// TIA Portal project "LAP_2018_Abfuellanlage" (V14)

(* hardware
DEVICE "S7-1200-Station_1"  S7-1200 Station
   slot 0: "Baugruppenträger_0"  S7-1200 Rack  Rack  V1.0
   slot 1: "PLC_1"  CPU 1214C DC/DC/DC  6ES7 214-1AG40-0XB0  V4.2
   slot 3: "AQ 1x12BIT_1"  AQ1 signal board  6ES7 232-4HA30-0XB0  V1.0
*)

// ===== PLC "PLC_1"  CPU 1214C DC/DC/DC =====

VAR_GLOBAL   // PLC tag table "Standard-Variablentabelle"
   "System_Byte" AT %MB100 : Byte;
   "FirstScan" AT %M100.0 : Bool;
   "DiagStatusUpdate" AT %M100.1 : Bool;
   "AlwaysTRUE" AT %M100.2 : Bool;
   "AlwaysFALSE" AT %M100.3 : Bool;
   "Clock_Byte" AT %MB110 : Byte;
   "Clock_10Hz" AT %M110.0 : Bool;
   "Clock_5Hz" AT %M110.1 : Bool;
   "Clock_2.5Hz" AT %M110.2 : Bool;
   "Clock_2Hz" AT %M110.3 : Bool;
   "Clock_1.25Hz" AT %M110.4 : Bool;
   "Clock_1Hz" AT %M110.5 : Bool;
   "Clock_0.625Hz" AT %M110.6 : Bool;
   "Clock_0.5Hz" AT %M110.7 : Bool;
   "Q1" AT %Q0.0 : Bool;   // Nicht verwenden! - Nur zum Testen
   "Q2" AT %Q0.1 : Bool;   // Nicht verwenden! - Nur zum Testen
   "S1" AT %I0.0 : Bool;   // Nicht verwenden! - Nur zum Testen
   "S2" AT %I0.1 : Bool;   // Nicht verwenden! - Nur zum Testen
   "S3" AT %I0.2 : Bool;   // Nicht verwenden! - Nur zum Testen
   "S4" AT %I0.3 : Bool;   // Nicht verwenden! - Nur zum Testen
   "S5" AT %I0.4 : Bool;   // Nicht verwenden! - Nur zum Testen
   "AlleAusgänge" AT %QW0 : Word;   // Nicht löschen!
   "Q3" AT %Q0.2 : Bool;   // Nicht verwenden! - Nur zum Testen
   "Q4" AT %Q0.3 : Bool;   // Nicht verwenden! - Nur zum Testen
   "Q5" AT %Q0.4 : Bool;   // Nicht verwenden! - Nur zum Testen
   "Q6" AT %Q0.5 : Bool;   // Nicht verwenden! - Nur zum Testen
END_VAR

DATA_BLOCK "VersionInput"   // DB1
{ S7_Optimized_Access := 'FALSE' }
VERSION : 0.1
   VAR
      AutoTest : Bool;
      "Version" : String := 'LAP 2018/2 Abfuellanlage V2.0';
   END_VAR
BEGIN
END_DATA_BLOCK

DATA_BLOCK "DigInput"   // DB2
{ S7_Optimized_Access := 'FALSE' }
VERSION : 0.1
   VAR
      B1 : Bool;   // Position Flasche
      F5 : Bool;   // Motorschutzschalter
      S1 : Bool;   // Start
      S2 : Bool;   // Stop
      S3 : Bool;   // Vereinzelung
      S4 : Bool;   // Quittieren
   END_VAR
BEGIN
END_DATA_BLOCK

DATA_BLOCK "DigOutput"   // DB3
{ S7_Optimized_Access := 'FALSE' }
VERSION : 0.1
   VAR
      M1 : Bool;   // Antrieb Förderband
      K1 : Bool;   // Füllung
      K2 : Bool;   // Vereinzelung
      P1 : Bool;   // Anlage Ein
      P2 : Bool;   // Störung
   END_VAR
BEGIN
END_DATA_BLOCK

DATA_BLOCK "AnInput"   // DB4
{ S7_Optimized_Access := 'FALSE' }
VERSION : 0.1
   VAR
      PegelByte : Byte;
      PegelInt : Int;
   END_VAR
BEGIN
END_DATA_BLOCK

FUNCTION "DeleteMe" : Void   // FC1, SCL
{ S7_Optimized_Access := 'TRUE' }
VERSION : 0.1
BEGIN
   "DigOutput".K1 := "S1";
   "DigOutput".K2 := "S2";
   "DigOutput".M1 := "S3";
   "DigOutput".P1 := "S4";
   "DigOutput".P2 := "S5";

   "Q1" := "DigInput".B1;
   "Q2" := "DigInput".F5;
   "Q3" := "DigInput".S1;
   "Q4" := "DigInput".S2;
   "Q5" := "DigInput".S3;
   "Q6" := "DigInput".S4;
END_FUNCTION

FUNCTION "DatenRangieren" : Void   // FC2, SCL
{ S7_Optimized_Access := 'TRUE' }
VERSION : 0.1
BEGIN
END_FUNCTION

ORGANIZATION_BLOCK "Main"   // OB1, LAD, ProgramCycle
TITLE = "Main Program Sweep (Cycle)"
{ S7_Optimized_Access := 'TRUE' }
VERSION : 0.1
   VAR_INPUT
      Initial_Call : Bool;   // Initial call of this OB
      Remanence : Bool;   // =True, if remanent data are available
   END_VAR
BEGIN

REGION Network 1
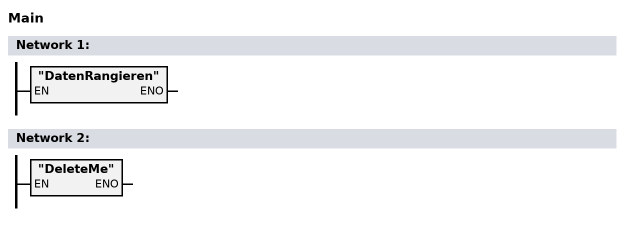
   RUNG wire#powerrail
      "DatenRangieren"()
   END_RUNG
   // the same network as SCL:
   "DatenRangieren"();
END_REGION

REGION Network 2
   RUNG wire#powerrail
      "DeleteMe"()
   END_RUNG
   // the same network as SCL:
   "DeleteMe"();
END_REGION
END_ORGANIZATION_BLOCK

ORGANIZATION_BLOCK "Startup"   // OB100, SCL, Startup
TITLE = "Complete Restart"
{ S7_Optimized_Access := 'TRUE' }
VERSION : 0.1
   VAR_INPUT
      LostRetentive : Bool;   // True if retentive data are lost
      LostRTC : Bool;   // True if date and time are lost
   END_VAR
BEGIN
   "AlleAusgänge" := 16#0000;
END_ORGANIZATION_BLOCK